KUKA KRL program: MillingProgram1.src, MillingProgram1.dat

--- MillingProgram1.src ---
&ACCESS RV
DEF MillingProgram1 ( )

END

--- MillingProgram1.dat ---
&ACCESS RV
DEFDAT MillingProgram1 PUBLIC

ENDDAT
